FUNCTION_BLOCK ConveyorCTLRingToken (* Basic Function Block Type *)
  (* Standard: 61499-2 *)
  (* Version 0.2, 2003-12-04, JHC, Rockwell Automation, Renamed for better indexing. *)
  (* Version 0.1, 2002-11-05, JHC, Rockwell Automation, Corrected missing ST element in Algorithm REQ. *)
  (* Version 0.0, 2000-05-30, JHC, Rockwell Automation *)
  (* Compiler header: package fb.rt.cs725; *)
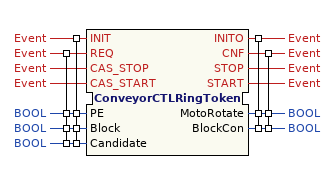
  EVENT_INPUT
    INIT WITH PE, Block, Candidate; (* Initialization Request *)
    REQ WITH PE, Block, Candidate; (* Normal Execution Request *)
    CAS_STOP;
    CAS_START;
  END_EVENT
  EVENT_OUTPUT
    INITO WITH MotoRotate, BlockCon; (* Initialization Confirm *)
    CNF WITH MotoRotate, BlockCon; (* Execution Confirmation *)
    STOP;
    START;
  END_EVENT
  VAR_INPUT
    PE : BOOL; (* Input event qualifier *)
    Block : BOOL;
    Candidate : BOOL;
  END_VAR
  VAR_OUTPUT
    MotoRotate : BOOL; (* Output event qualifier *)
    BlockCon : BOOL;
  END_VAR
  VAR
    lastPE : BOOL := 1;
    lastBlock : BOOL := 0;
  END_VAR
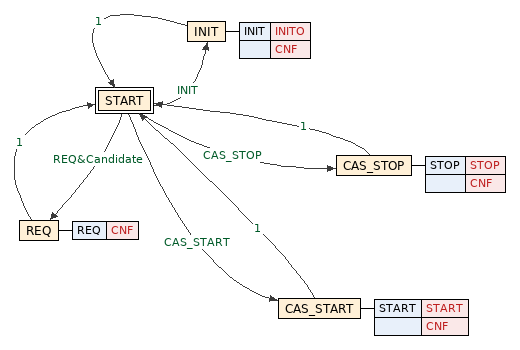
  EC_STATES
    START; (* Initial State *)
    INIT : INIT -> INITO, -> CNF; (* Initialization *)
    REQ : REQ -> CNF; (* Normal execution *)
    CAS_START : START -> START, -> CNF;
    CAS_STOP : STOP -> STOP, -> CNF;
  END_STATES
  EC_TRANSITIONS
    START TO INIT := INIT;
    INIT TO START := 1;
    START TO REQ := REQ&Candidate;
    REQ TO START := 1;
    START TO CAS_START := CAS_START;
    CAS_START TO START := 1;
    START TO CAS_STOP := CAS_STOP;
    CAS_STOP TO START := 1;
  END_TRANSITIONS
  ALGORITHM INIT IN ST: (* Initialization algorithm *)
MotoRotate := TRUE;
Block := FALSE;

System.out.println(this + " " + MotoRotate);
System.out.println(MotoRotate);
  END_ALGORITHM
  ALGORITHM REQ IN ST: (* Normally executed algorithm *)
System.out.println(this +  " -> Candidate" + Candidate);
IF Candidate THEN
IF lastPE !:= PE THEN
IF NOT PE THEN
BlockCon:= TRUE;
System.out.println("BlockCon = true");
ELSE
BlockCon:=FALSE;
System.out.println("BlockCon = false");
END_IF
lastPE := PE;
END_IF
IF lastBlock !:= Block THEN
IF Block THEN
STOP.serviceEvent(this);
MotoRotate := FALSE;
System.out.println("Cas Stop");
ELSE
START.serviceEvent(this);
MotoRotate := TRUE;
System.out.println("Cas Start");
END_IF
lastBlock := Block;
END_IF
END_IF
  END_ALGORITHM
  ALGORITHM START IN ST:
MotoRotate:=TRUE;
System.out.println(this + " Start " + MotoRotate);

System.out.println("Start " + MotoRotate);
  END_ALGORITHM
  ALGORITHM STOP IN ST:
MotoRotate := FALSE;
System.out.println(this + " Stop " + MotoRotate);

System.out.println("Stop " + MotoRotate);
  END_ALGORITHM
END_FUNCTION_BLOCK
